% RSLogix 500 project EDINBURG_BAK719.RSS, saved by version 10.00.00.00 %
PROJECT "EDINBURG"    % processor: MicroLogix 1400 %

PROGRAM FILES
  LAD 2   12 rungs
  LAD 3   11 rungs
  LAD 4   11 rungs
  LAD 5   25 rungs
  LAD 6   8 rungs
  LAD 7   17 rungs
  LAD 8   4 rungs
  LAD 9   35 rungs
  LAD 10   2 rungs
  LAD 11   49 rungs
  LAD 12   13 rungs
  LAD 13   23 rungs

DATA FILES
  O0 OUTPUT  9 elements
  I1 INPUT  11 elements
  S2 STATUS  66 elements
  B3 BINARY  7 elements
  T4 TIMER  38 elements
  C5 COUNTER  1 elements
  R6 CONTROL  1 elements
  N7 INTEGER  40 elements
  F8 FLOAT  30 elements
  L9   1 elements
  L10   2 elements

LADDER 2
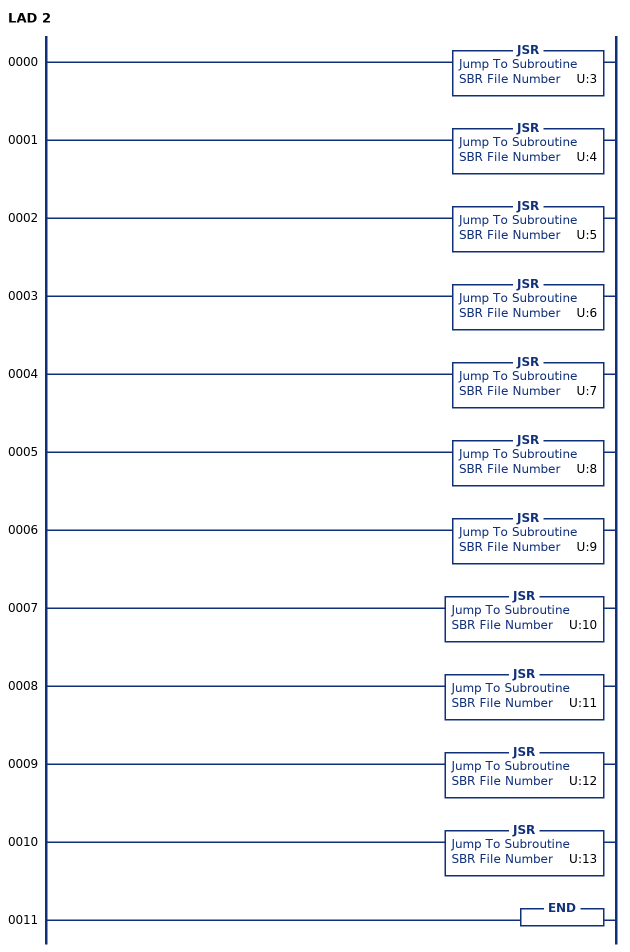
% Rung: 0 %
SOR JSR U:3 EOR
% Rung: 1 %
SOR JSR U:4 EOR
% Rung: 2 %
SOR JSR U:5 EOR
% Rung: 3 %
SOR JSR U:6 EOR
% Rung: 4 %
SOR JSR U:7 EOR
% Rung: 5 %
SOR JSR U:8 EOR
% Rung: 6 %
SOR JSR U:9 EOR
% Rung: 7 %
SOR JSR U:10 EOR
% Rung: 8 %
SOR JSR U:11 EOR
% Rung: 9 %
SOR JSR U:12 EOR
% Rung: 10 %
SOR JSR U:13 EOR
% Rung: 11 %
SOR END EOR

LADDER 3
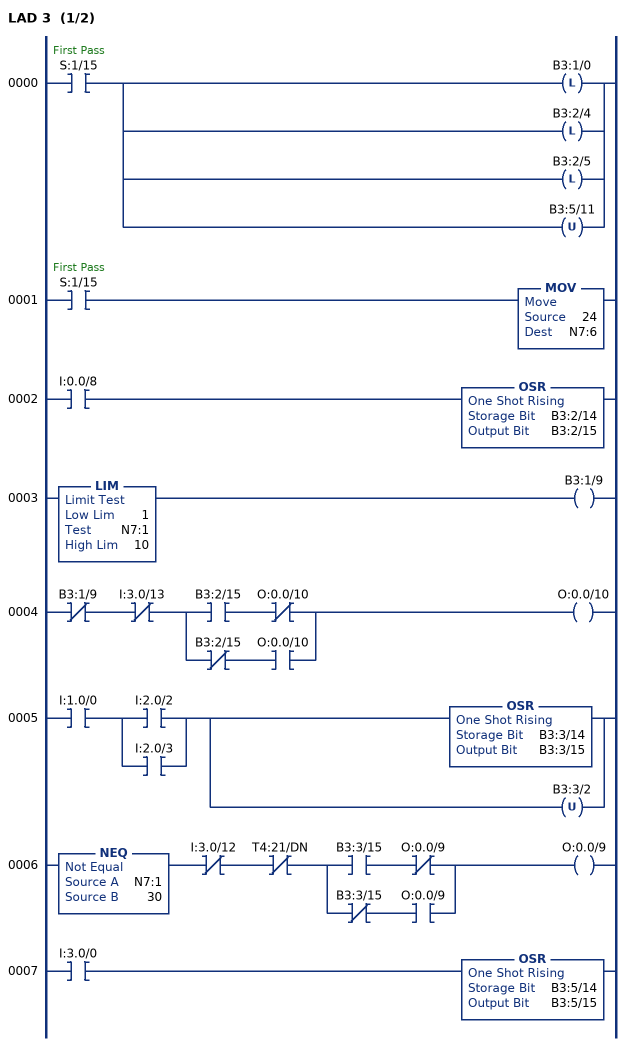
% Rung: 0 %
SOR XIC S:1/15 BST OTL B3:1/0 NXB BST OTL B3:2/4 NXB BST OTL B3:2/5 NXB OTU B3:5/11 BND BND BND EOR
%   S:1/15  "First Pass" %
% Rung: 1 %
SOR XIC S:1/15 MOV 24 N7:6 EOR
%   S:1/15  "First Pass" %
% Rung: 2 %
SOR XIC I:0.0/8 OSR B3:2/14 B3:2/15 EOR
% Rung: 3 %
SOR LIM 1 N7:1 10 OTE B3:1/9 EOR
% Rung: 4 %
SOR XIO B3:1/9 XIO I:3.0/13 BST XIC B3:2/15 XIO O:0.0/10 NXB XIO B3:2/15 XIC O:0.0/10 BND OTE O:0.0/10 EOR
% Rung: 5 %
SOR XIC I:1.0/0 BST XIC I:2.0/2 NXB XIC I:2.0/3 BND BST OSR B3:3/14 B3:3/15 NXB OTU B3:3/2 BND EOR
% Rung: 6 %
SOR NEQ N7:1 30 XIO I:3.0/12 XIO T4:21/DN BST XIC B3:3/15 XIO O:0.0/9 NXB XIO B3:3/15 XIC O:0.0/9 BND OTE O:0.0/9 EOR
% Rung: 7 %
SOR XIC I:3.0/0 OSR B3:5/14 B3:5/15 EOR

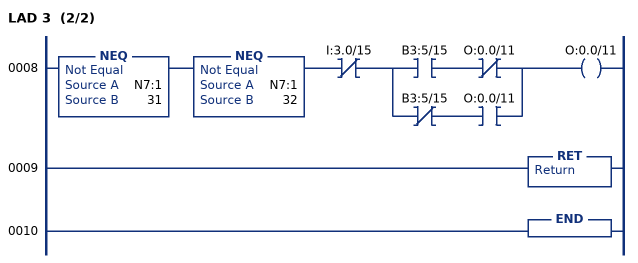
% Rung: 8 %
SOR NEQ N7:1 31 NEQ N7:1 32 XIO I:3.0/15 BST XIC B3:5/15 XIO O:0.0/11 NXB XIO B3:5/15 XIC O:0.0/11 BND OTE O:0.0/11 EOR
% Rung: 9 %
SOR RET EOR
% Rung: 10 %
SOR END EOR

LADDER 4
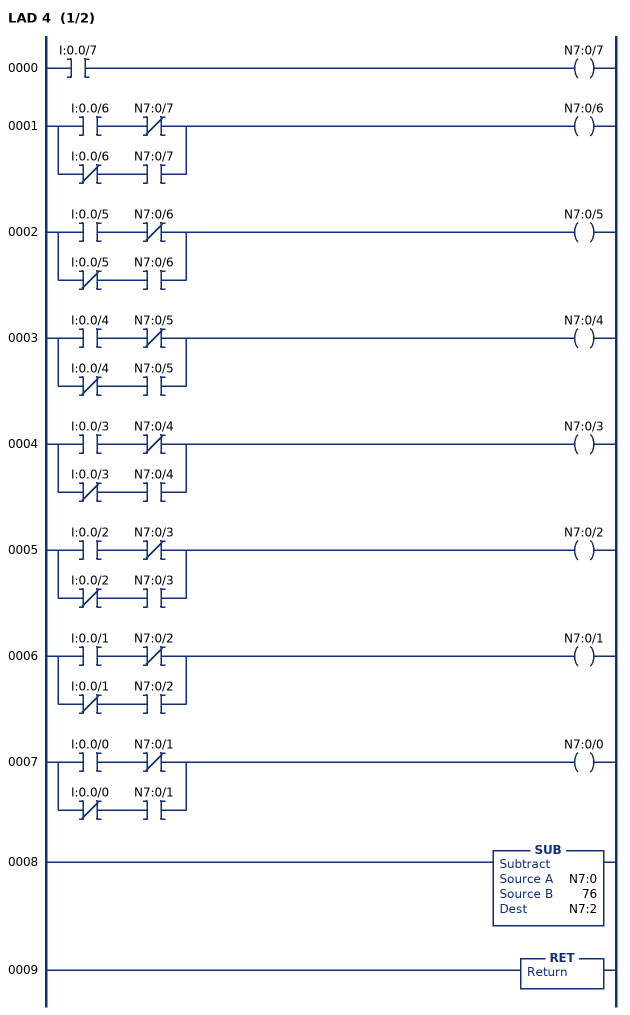
% Rung: 0 %
SOR XIC I:0.0/7 OTE N7:0/7 EOR
% Rung: 1 %
SOR BST XIC I:0.0/6 XIO N7:0/7 NXB XIO I:0.0/6 XIC N7:0/7 BND OTE N7:0/6 EOR
% Rung: 2 %
SOR BST XIC I:0.0/5 XIO N7:0/6 NXB XIO I:0.0/5 XIC N7:0/6 BND OTE N7:0/5 EOR
% Rung: 3 %
SOR BST XIC I:0.0/4 XIO N7:0/5 NXB XIO I:0.0/4 XIC N7:0/5 BND OTE N7:0/4 EOR
% Rung: 4 %
SOR BST XIC I:0.0/3 XIO N7:0/4 NXB XIO I:0.0/3 XIC N7:0/4 BND OTE N7:0/3 EOR
% Rung: 5 %
SOR BST XIC I:0.0/2 XIO N7:0/3 NXB XIO I:0.0/2 XIC N7:0/3 BND OTE N7:0/2 EOR
% Rung: 6 %
SOR BST XIC I:0.0/1 XIO N7:0/2 NXB XIO I:0.0/1 XIC N7:0/2 BND OTE N7:0/1 EOR
% Rung: 7 %
SOR BST XIC I:0.0/0 XIO N7:0/1 NXB XIO I:0.0/0 XIC N7:0/1 BND OTE N7:0/0 EOR
% Rung: 8 %
SOR SUB N7:0 76 N7:2 EOR
% Rung: 9 %
SOR RET EOR

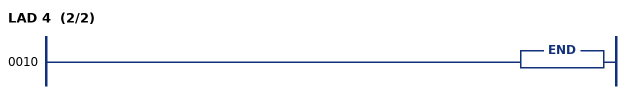
% Rung: 10 %
SOR END EOR

LADDER 5
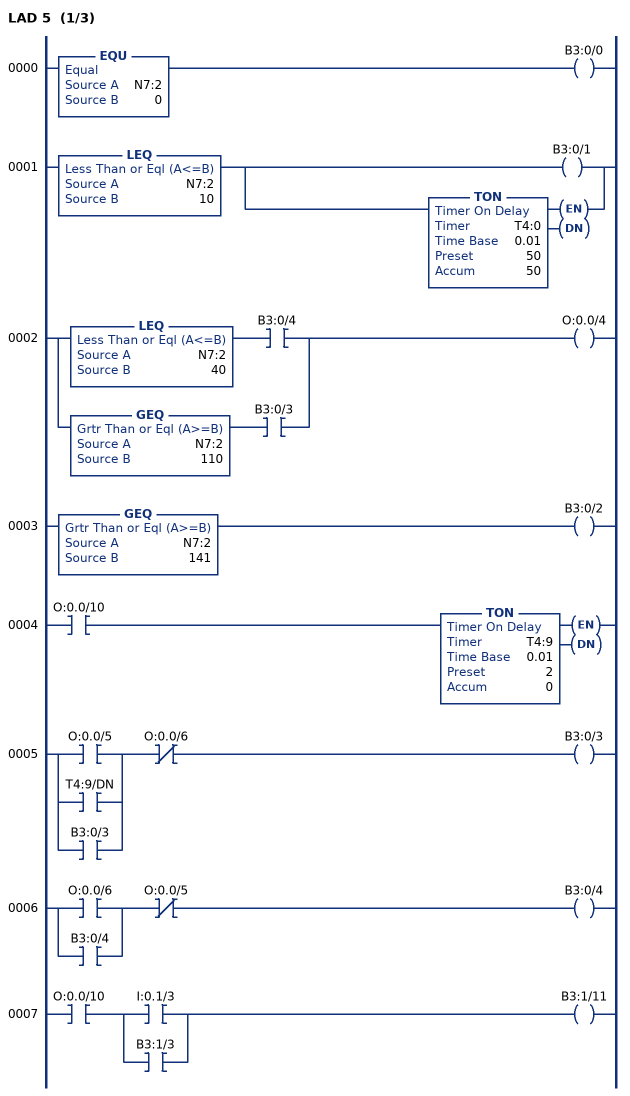
% Rung: 0 %
SOR EQU N7:2 0 OTE B3:0/0 EOR
% Rung: 1 %
SOR LEQ N7:2 10 BST OTE B3:0/1 NXB TON T4:0 0.01 50 50 BND EOR
% Rung: 2 %
SOR BST LEQ N7:2 40 XIC B3:0/4 NXB GEQ N7:2 110 XIC B3:0/3 BND OTE O:0.0/4 EOR
% Rung: 3 %
SOR GEQ N7:2 141 OTE B3:0/2 EOR
% Rung: 4 %
SOR XIC O:0.0/10 TON T4:9 0.01 2 0 EOR
% Rung: 5 %
SOR BST XIC O:0.0/5 NXB XIC T4:9/DN NXB XIC B3:0/3 BND XIO O:0.0/6 OTE B3:0/3 EOR
% Rung: 6 %
SOR BST XIC O:0.0/6 NXB XIC B3:0/4 BND XIO O:0.0/5 OTE B3:0/4 EOR
% Rung: 7 %
SOR XIC O:0.0/10 BST XIC I:0.1/3 NXB XIC B3:1/3 BND OTE B3:1/11 EOR

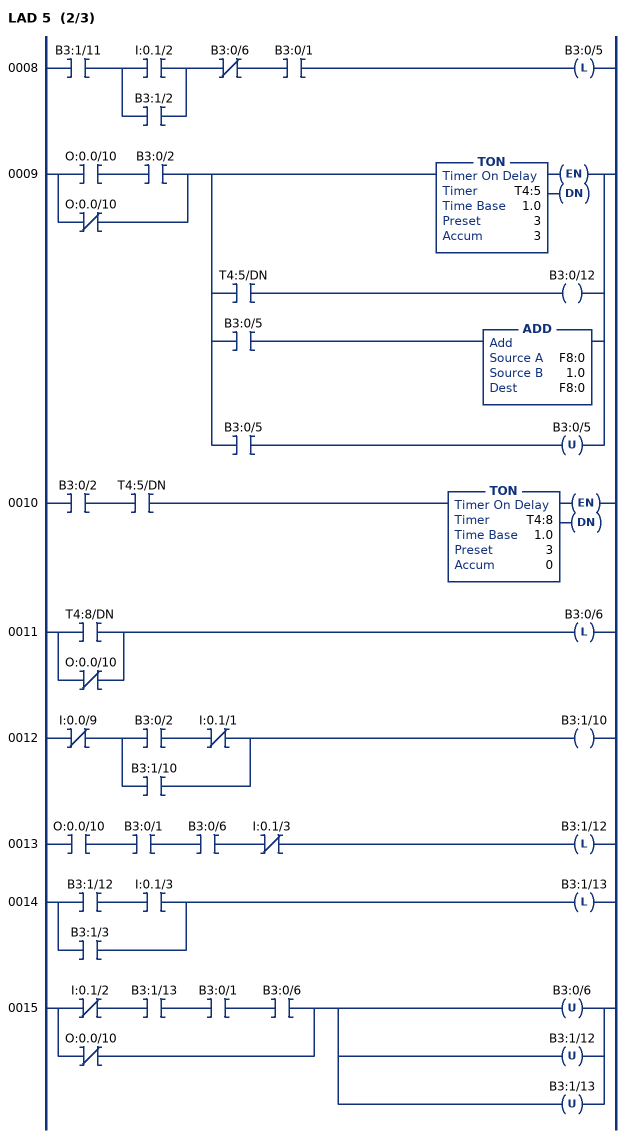
% Rung: 8 %
SOR XIC B3:1/11 BST XIC I:0.1/2 NXB XIC B3:1/2 BND XIO B3:0/6 XIC B3:0/1 OTL B3:0/5 EOR
% Rung: 9 %
SOR BST XIC O:0.0/10 XIC B3:0/2 NXB XIO O:0.0/10 BND BST TON T4:5 1.0 3 3 NXB XIC T4:5/DN OTE B3:0/12 NXB BST XIC B3:0/5 ADD F8:0 1.0 F8:0 NXB XIC B3:0/5 OTU B3:0/5 BND BND EOR
% Rung: 10 %
SOR XIC B3:0/2 XIC T4:5/DN TON T4:8 1.0 3 0 EOR
% Rung: 11 %
SOR BST XIC T4:8/DN NXB XIO O:0.0/10 BND OTL B3:0/6 EOR
% Rung: 12 %
SOR XIO I:0.0/9 BST XIC B3:0/2 XIO I:0.1/1 NXB XIC B3:1/10 BND OTE B3:1/10 EOR
% Rung: 13 %
SOR XIC O:0.0/10 XIC B3:0/1 XIC B3:0/6 XIO I:0.1/3 OTL B3:1/12 EOR
% Rung: 14 %
SOR BST XIC B3:1/12 XIC I:0.1/3 NXB XIC B3:1/3 BND OTL B3:1/13 EOR
% Rung: 15 %
SOR BST XIO I:0.1/2 XIC B3:1/13 XIC B3:0/1 XIC B3:0/6 NXB XIO O:0.0/10 BND BST OTU B3:0/6 NXB BST OTU B3:1/12 NXB OTU B3:1/13 BND BND EOR

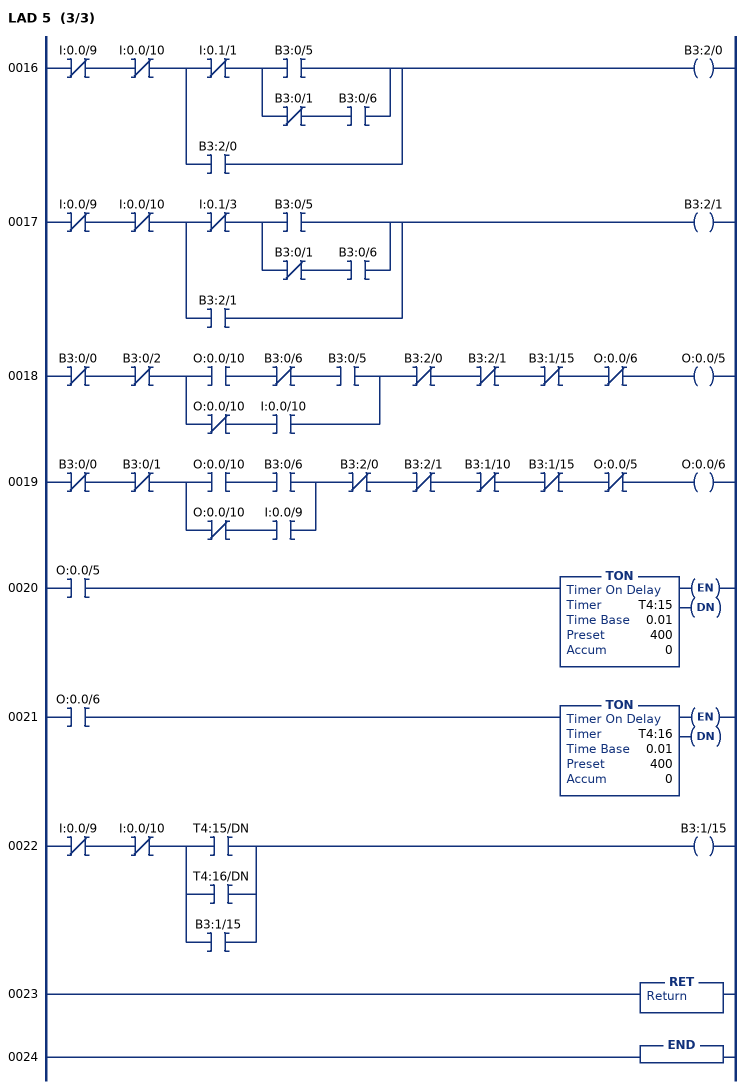
% Rung: 16 %
SOR XIO I:0.0/9 XIO I:0.0/10 BST XIO I:0.1/1 BST XIC B3:0/5 NXB XIO B3:0/1 XIC B3:0/6 BND NXB XIC B3:2/0 BND OTE B3:2/0 EOR
% Rung: 17 %
SOR XIO I:0.0/9 XIO I:0.0/10 BST XIO I:0.1/3 BST XIC B3:0/5 NXB XIO B3:0/1 XIC B3:0/6 BND NXB XIC B3:2/1 BND OTE B3:2/1 EOR
% Rung: 18 %
SOR XIO B3:0/0 XIO B3:0/2 BST XIC O:0.0/10 XIO B3:0/6 XIC B3:0/5 NXB XIO O:0.0/10 XIC I:0.0/10 BND XIO B3:2/0 XIO B3:2/1 XIO B3:1/15 XIO O:0.0/6 OTE O:0.0/5 EOR
% Rung: 19 %
SOR XIO B3:0/0 XIO B3:0/1 BST XIC O:0.0/10 XIC B3:0/6 NXB XIO O:0.0/10 XIC I:0.0/9 BND XIO B3:2/0 XIO B3:2/1 XIO B3:1/10 XIO B3:1/15 XIO O:0.0/5 OTE O:0.0/6 EOR
% Rung: 20 %
SOR XIC O:0.0/5 TON T4:15 0.01 400 0 EOR
% Rung: 21 %
SOR XIC O:0.0/6 TON T4:16 0.01 400 0 EOR
% Rung: 22 %
SOR XIO I:0.0/9 XIO I:0.0/10 BST BST XIC T4:15/DN NXB XIC T4:16/DN BND NXB XIC B3:1/15 BND OTE B3:1/15 EOR
% Rung: 23 %
SOR RET EOR
% Rung: 24 %
SOR END EOR

LADDER 6
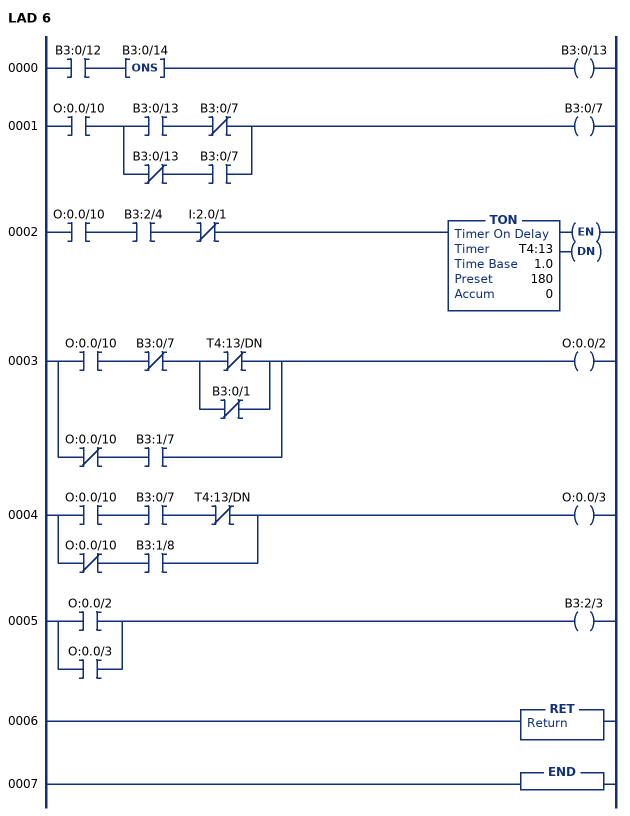
% Rung: 0 %
SOR XIC B3:0/12 ONS B3:0/14 OTE B3:0/13 EOR
% Rung: 1 %
SOR XIC O:0.0/10 BST XIC B3:0/13 XIO B3:0/7 NXB XIO B3:0/13 XIC B3:0/7 BND OTE B3:0/7 EOR
% Rung: 2 %
SOR XIC O:0.0/10 XIC B3:2/4 XIO I:2.0/1 TON T4:13 1.0 180 0 EOR
% Rung: 3 %
SOR BST XIC O:0.0/10 XIO B3:0/7 BST XIO T4:13/DN NXB XIO B3:0/1 BND NXB XIO O:0.0/10 XIC B3:1/7 BND OTE O:0.0/2 EOR
% Rung: 4 %
SOR BST XIC O:0.0/10 XIC B3:0/7 XIO T4:13/DN NXB XIO O:0.0/10 XIC B3:1/8 BND OTE O:0.0/3 EOR
% Rung: 5 %
SOR BST XIC O:0.0/2 NXB XIC O:0.0/3 BND OTE B3:2/3 EOR
% Rung: 6 %
SOR RET EOR
% Rung: 7 %
SOR END EOR

LADDER 7
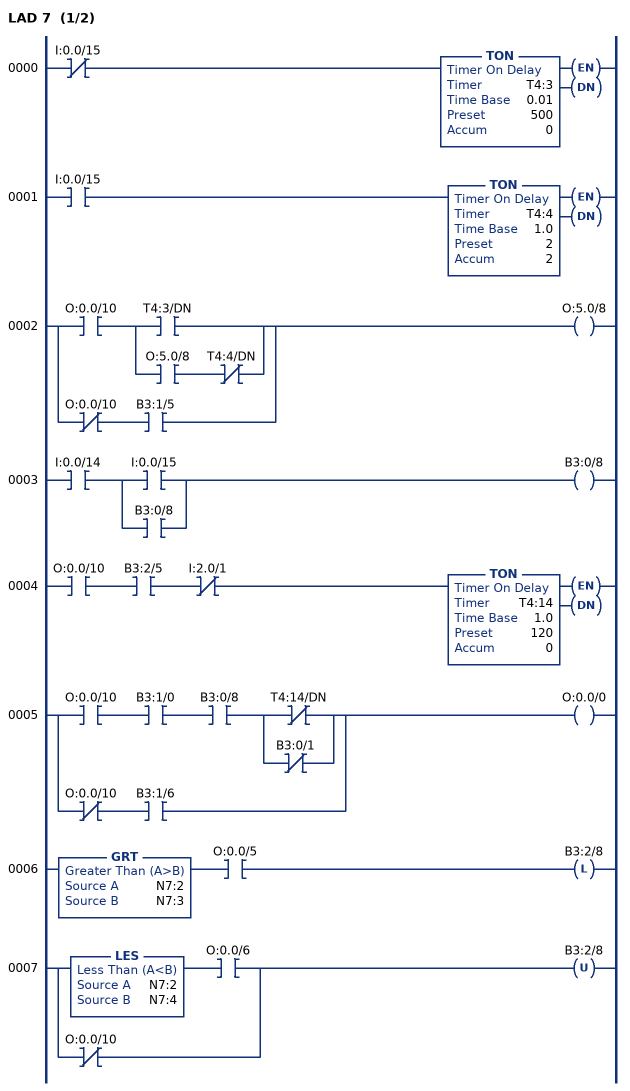
% Rung: 0 %
SOR XIO I:0.0/15 TON T4:3 0.01 500 0 EOR
% Rung: 1 %
SOR XIC I:0.0/15 TON T4:4 1.0 2 2 EOR
% Rung: 2 %
SOR BST XIC O:0.0/10 BST XIC T4:3/DN NXB XIC O:5.0/8 XIO T4:4/DN BND NXB XIO O:0.0/10 XIC B3:1/5 BND OTE O:5.0/8 EOR
% Rung: 3 %
SOR XIC I:0.0/14 BST XIC I:0.0/15 NXB XIC B3:0/8 BND OTE B3:0/8 EOR
% Rung: 4 %
SOR XIC O:0.0/10 XIC B3:2/5 XIO I:2.0/1 TON T4:14 1.0 120 0 EOR
% Rung: 5 %
SOR BST XIC O:0.0/10 XIC B3:1/0 XIC B3:0/8 BST XIO T4:14/DN NXB XIO B3:0/1 BND NXB XIO O:0.0/10 XIC B3:1/6 BND OTE O:0.0/0 EOR
% Rung: 6 %
SOR GRT N7:2 N7:3 XIC O:0.0/5 OTL B3:2/8 EOR
% Rung: 7 %
SOR BST LES N7:2 N7:4 XIC O:0.0/6 NXB XIO O:0.0/10 BND OTU B3:2/8 EOR

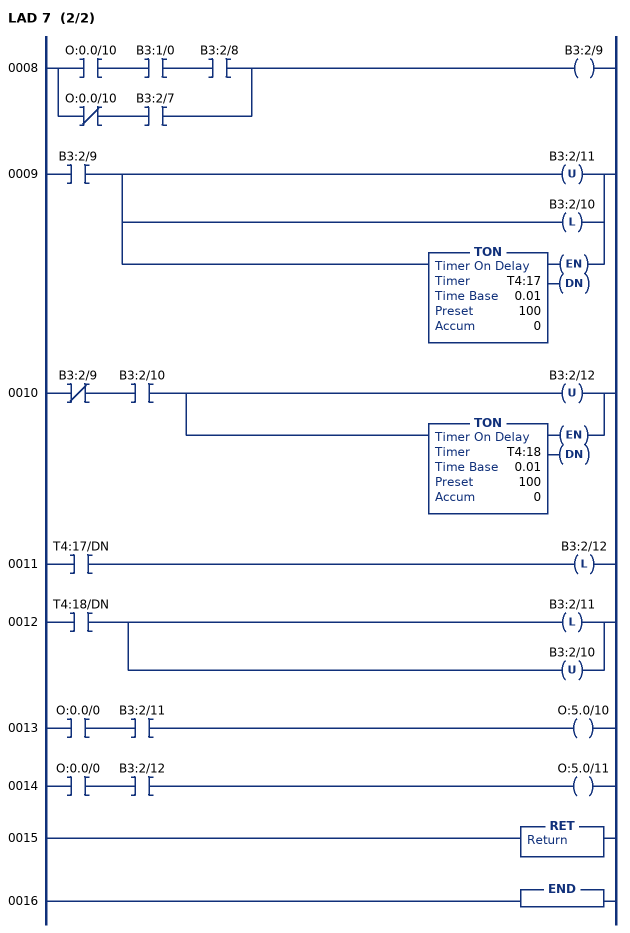
% Rung: 8 %
SOR BST XIC O:0.0/10 XIC B3:1/0 XIC B3:2/8 NXB XIO O:0.0/10 XIC B3:2/7 BND OTE B3:2/9 EOR
% Rung: 9 %
SOR XIC B3:2/9 BST OTU B3:2/11 NXB BST OTL B3:2/10 NXB TON T4:17 0.01 100 0 BND BND EOR
% Rung: 10 %
SOR XIO B3:2/9 XIC B3:2/10 BST OTU B3:2/12 NXB TON T4:18 0.01 100 0 BND EOR
% Rung: 11 %
SOR XIC T4:17/DN OTL B3:2/12 EOR
% Rung: 12 %
SOR XIC T4:18/DN BST OTL B3:2/11 NXB OTU B3:2/10 BND EOR
% Rung: 13 %
SOR XIC O:0.0/0 XIC B3:2/11 OTE O:5.0/10 EOR
% Rung: 14 %
SOR XIC O:0.0/0 XIC B3:2/12 OTE O:5.0/11 EOR
% Rung: 15 %
SOR RET EOR
% Rung: 16 %
SOR END EOR

LADDER 8
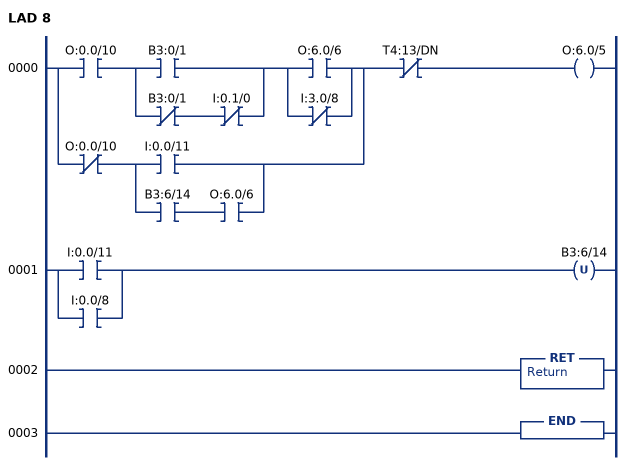
% Rung: 0 %
SOR BST XIC O:0.0/10 BST XIC B3:0/1 NXB XIO B3:0/1 XIO I:0.1/0 BND BST XIC O:6.0/6 NXB XIO I:3.0/8 BND NXB XIO O:0.0/10 BST XIC I:0.0/11 NXB XIC B3:6/14 XIC O:6.0/6 BND BND XIO T4:13/DN OTE O:6.0/5 EOR
% Rung: 1 %
SOR BST XIC I:0.0/11 NXB XIC I:0.0/8 BND OTU B3:6/14 EOR
% Rung: 2 %
SOR RET EOR
% Rung: 3 %
SOR END EOR

LADDER 9
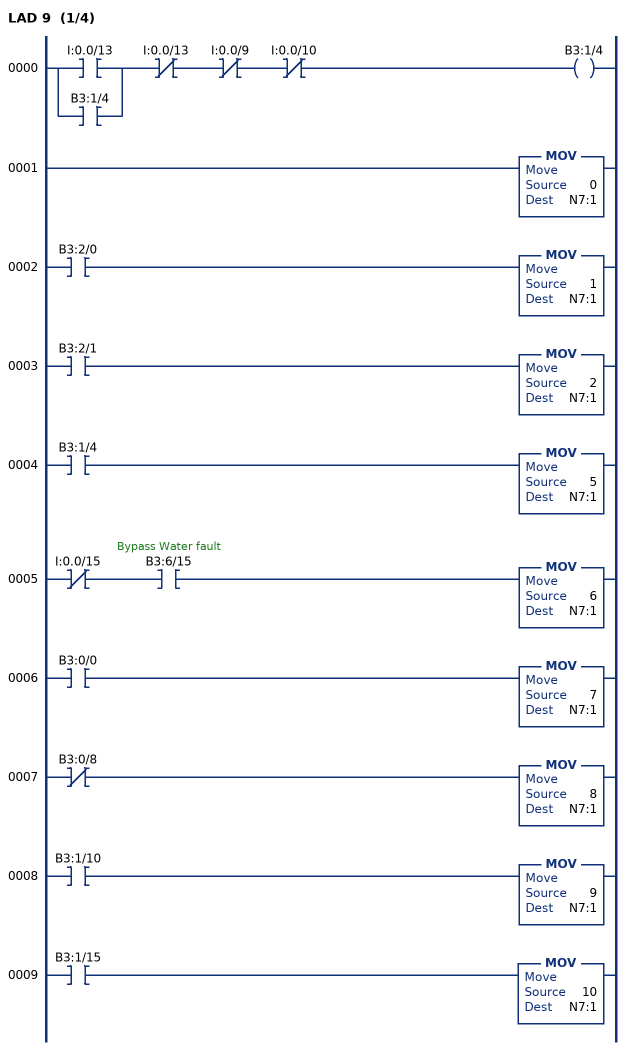
% Rung: 0 %
SOR BST XIC I:0.0/13 NXB XIC B3:1/4 BND XIO I:0.0/13 XIO I:0.0/9 XIO I:0.0/10 OTE B3:1/4 EOR
% Rung: 1 %
SOR MOV 0 N7:1 EOR
% Rung: 2 %
SOR XIC B3:2/0 MOV 1 N7:1 EOR
% Rung: 3 %
SOR XIC B3:2/1 MOV 2 N7:1 EOR
% Rung: 4 %
SOR XIC B3:1/4 MOV 5 N7:1 EOR
% Rung: 5 %
SOR XIO I:0.0/15 XIC B3:6/15 MOV 6 N7:1 EOR
%   B3:6/15  "Bypass Water fault" %
% Rung: 6 %
SOR XIC B3:0/0 MOV 7 N7:1 EOR
% Rung: 7 %
SOR XIO B3:0/8 MOV 8 N7:1 EOR
% Rung: 8 %
SOR XIC B3:1/10 MOV 9 N7:1 EOR
% Rung: 9 %
SOR XIC B3:1/15 MOV 10 N7:1 EOR

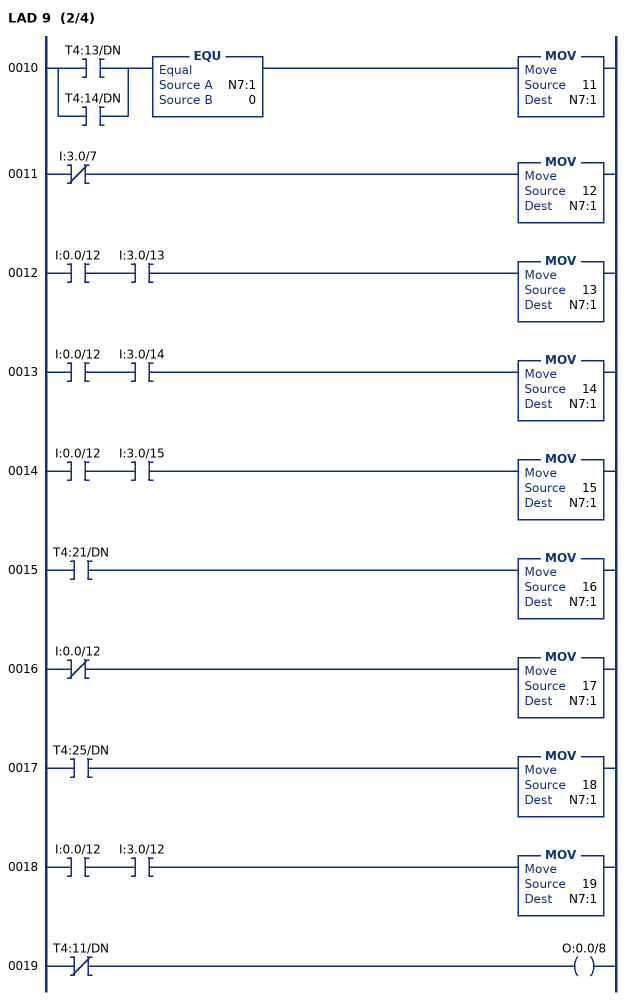
% Rung: 10 %
SOR BST XIC T4:13/DN NXB XIC T4:14/DN BND EQU N7:1 0 MOV 11 N7:1 EOR
% Rung: 11 %
SOR XIO I:3.0/7 MOV 12 N7:1 EOR
% Rung: 12 %
SOR XIC I:0.0/12 XIC I:3.0/13 MOV 13 N7:1 EOR
% Rung: 13 %
SOR XIC I:0.0/12 XIC I:3.0/14 MOV 14 N7:1 EOR
% Rung: 14 %
SOR XIC I:0.0/12 XIC I:3.0/15 MOV 15 N7:1 EOR
% Rung: 15 %
SOR XIC T4:21/DN MOV 16 N7:1 EOR
% Rung: 16 %
SOR XIO I:0.0/12 MOV 17 N7:1 EOR
% Rung: 17 %
SOR XIC T4:25/DN MOV 18 N7:1 EOR
% Rung: 18 %
SOR XIC I:0.0/12 XIC I:3.0/12 MOV 19 N7:1 EOR
% Rung: 19 %
SOR XIO T4:11/DN OTE O:0.0/8 EOR

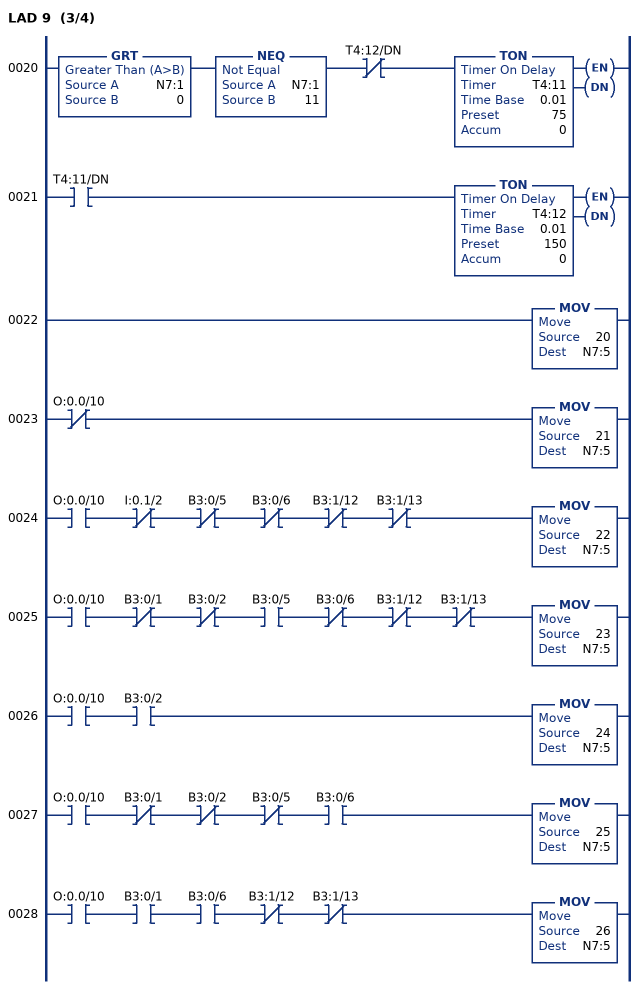
% Rung: 20 %
SOR GRT N7:1 0 NEQ N7:1 11 XIO T4:12/DN TON T4:11 0.01 75 0 EOR
% Rung: 21 %
SOR XIC T4:11/DN TON T4:12 0.01 150 0 EOR
% Rung: 22 %
SOR MOV 20 N7:5 EOR
% Rung: 23 %
SOR XIO O:0.0/10 MOV 21 N7:5 EOR
% Rung: 24 %
SOR XIC O:0.0/10 XIO I:0.1/2 XIO B3:0/5 XIO B3:0/6 XIO B3:1/12 XIO B3:1/13 MOV 22 N7:5 EOR
% Rung: 25 %
SOR XIC O:0.0/10 XIO B3:0/1 XIO B3:0/2 XIC B3:0/5 XIO B3:0/6 XIO B3:1/12 XIO B3:1/13 MOV 23 N7:5 EOR
% Rung: 26 %
SOR XIC O:0.0/10 XIC B3:0/2 MOV 24 N7:5 EOR
% Rung: 27 %
SOR XIC O:0.0/10 XIO B3:0/1 XIO B3:0/2 XIO B3:0/5 XIC B3:0/6 MOV 25 N7:5 EOR
% Rung: 28 %
SOR XIC O:0.0/10 XIC B3:0/1 XIC B3:0/6 XIO B3:1/12 XIO B3:1/13 MOV 26 N7:5 EOR

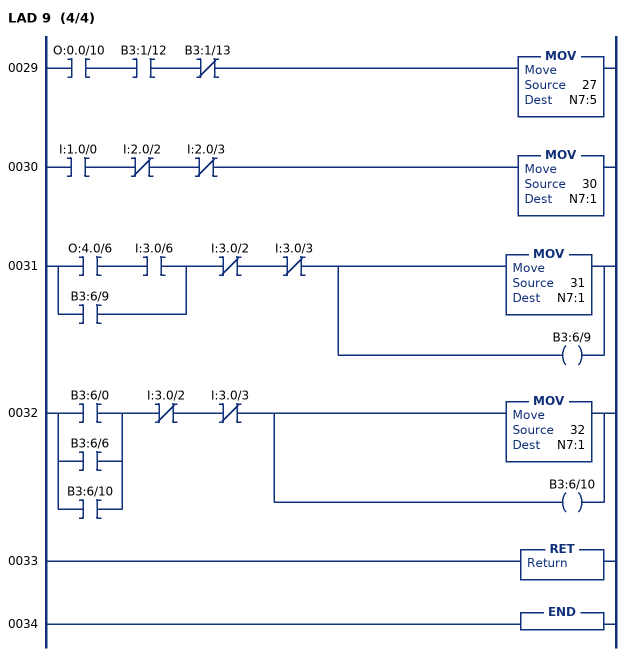
% Rung: 29 %
SOR XIC O:0.0/10 XIC B3:1/12 XIO B3:1/13 MOV 27 N7:5 EOR
% Rung: 30 %
SOR XIC I:1.0/0 XIO I:2.0/2 XIO I:2.0/3 MOV 30 N7:1 EOR
% Rung: 31 %
SOR BST XIC O:4.0/6 XIC I:3.0/6 NXB XIC B3:6/9 BND XIO I:3.0/2 XIO I:3.0/3 BST MOV 31 N7:1 NXB OTE B3:6/9 BND EOR
% Rung: 32 %
SOR BST BST XIC B3:6/0 NXB XIC B3:6/6 BND NXB XIC B3:6/10 BND XIO I:3.0/2 XIO I:3.0/3 BST MOV 32 N7:1 NXB OTE B3:6/10 BND EOR
% Rung: 33 %
SOR RET EOR
% Rung: 34 %
SOR END EOR

LADDER 10
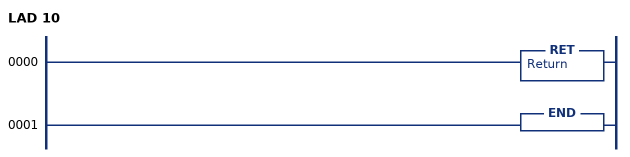
% Rung: 0 %
SOR RET EOR
% Rung: 1 %
SOR END EOR

LADDER 11
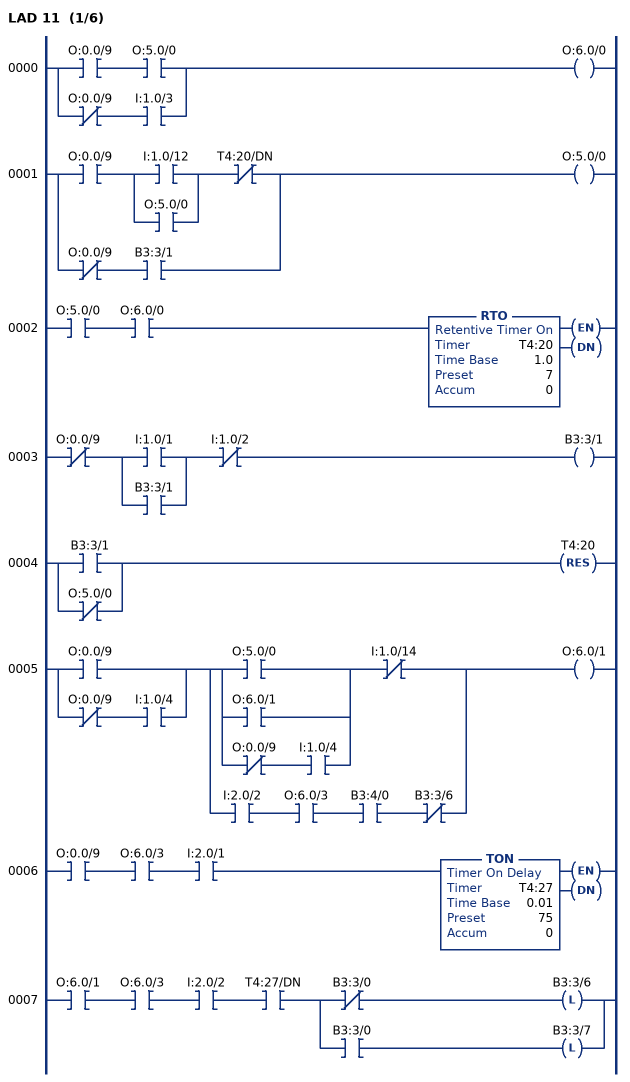
% Rung: 0 %
SOR BST XIC O:0.0/9 XIC O:5.0/0 NXB XIO O:0.0/9 XIC I:1.0/3 BND OTE O:6.0/0 EOR
% Rung: 1 %
SOR BST XIC O:0.0/9 BST XIC I:1.0/12 NXB XIC O:5.0/0 BND XIO T4:20/DN NXB XIO O:0.0/9 XIC B3:3/1 BND OTE O:5.0/0 EOR
% Rung: 2 %
SOR XIC O:5.0/0 XIC O:6.0/0 RTO T4:20 1.0 7 0 EOR
% Rung: 3 %
SOR XIO O:0.0/9 BST XIC I:1.0/1 NXB XIC B3:3/1 BND XIO I:1.0/2 OTE B3:3/1 EOR
% Rung: 4 %
SOR BST XIC B3:3/1 NXB XIO O:5.0/0 BND RES T4:20 EOR
% Rung: 5 %
SOR BST XIC O:0.0/9 NXB XIO O:0.0/9 XIC I:1.0/4 BND BST BST XIC O:5.0/0 NXB BST XIC O:6.0/1 NXB XIO O:0.0/9 XIC I:1.0/4 BND BND XIO I:1.0/14 NXB XIC I:2.0/2 XIC O:6.0/3 XIC B3:4/0 XIO B3:3/6 BND OTE O:6.0/1 EOR
% Rung: 6 %
SOR XIC O:0.0/9 XIC O:6.0/3 XIC I:2.0/1 TON T4:27 0.01 75 0 EOR
% Rung: 7 %
SOR XIC O:6.0/1 XIC O:6.0/3 XIC I:2.0/2 XIC T4:27/DN BST XIO B3:3/0 OTL B3:3/6 NXB XIC B3:3/0 OTL B3:3/7 BND EOR

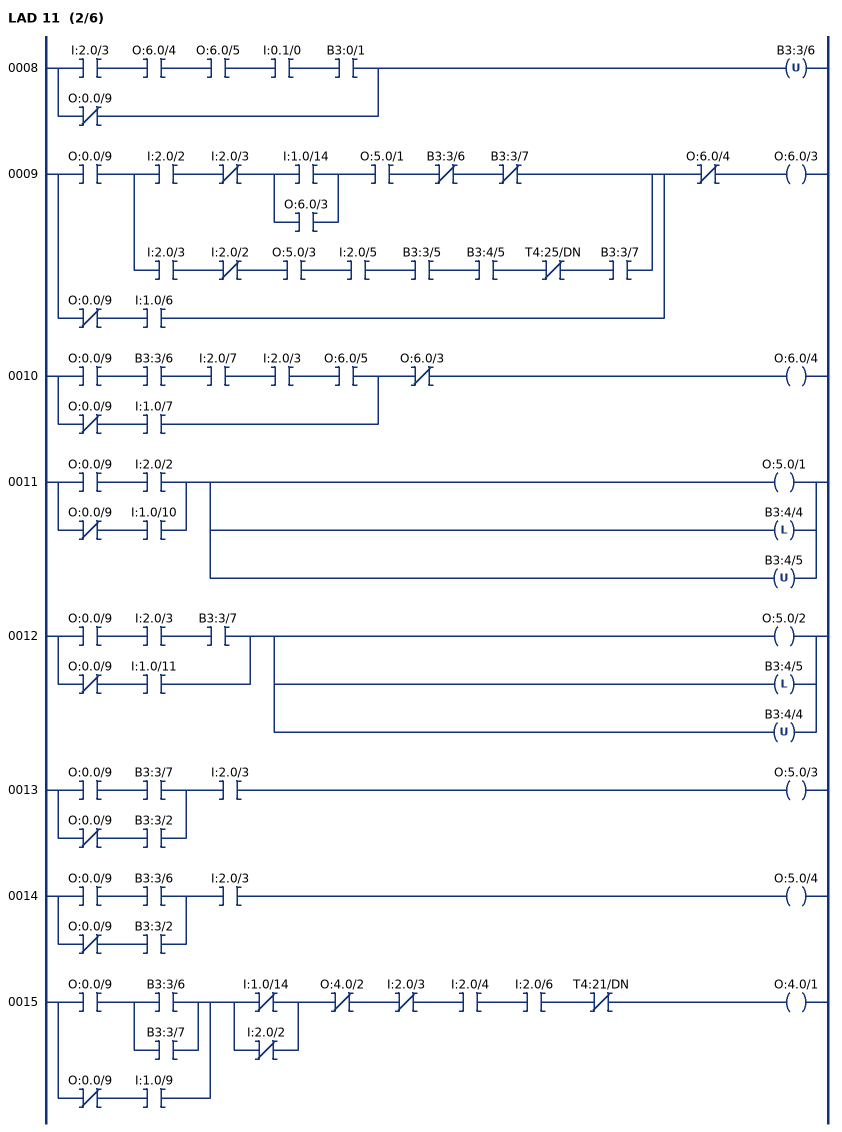
% Rung: 8 %
SOR BST XIC I:2.0/3 XIC O:6.0/4 XIC O:6.0/5 XIC I:0.1/0 XIC B3:0/1 NXB XIO O:0.0/9 BND OTU B3:3/6 EOR
% Rung: 9 %
SOR BST XIC O:0.0/9 BST XIC I:2.0/2 XIO I:2.0/3 BST XIC I:1.0/14 NXB XIC O:6.0/3 BND XIC O:5.0/1 XIO B3:3/6 XIO B3:3/7 NXB XIC I:2.0/3 XIO I:2.0/2 XIC O:5.0/3 XIC I:2.0/5 XIC B3:3/5 XIC B3:4/5 XIO T4:25/DN XIC B3:3/7 BND NXB XIO O:0.0/9 XIC I:1.0/6 BND XIO O:6.0/4 OTE O:6.0/3 EOR
% Rung: 10 %
SOR BST XIC O:0.0/9 XIC B3:3/6 XIC I:2.0/7 XIC I:2.0/3 XIC O:6.0/5 NXB XIO O:0.0/9 XIC I:1.0/7 BND XIO O:6.0/3 OTE O:6.0/4 EOR
% Rung: 11 %
SOR BST XIC O:0.0/9 XIC I:2.0/2 NXB XIO O:0.0/9 XIC I:1.0/10 BND BST OTE O:5.0/1 NXB BST OTL B3:4/4 NXB OTU B3:4/5 BND BND EOR
% Rung: 12 %
SOR BST XIC O:0.0/9 XIC I:2.0/3 XIC B3:3/7 NXB XIO O:0.0/9 XIC I:1.0/11 BND BST OTE O:5.0/2 NXB BST OTL B3:4/5 NXB OTU B3:4/4 BND BND EOR
% Rung: 13 %
SOR BST XIC O:0.0/9 XIC B3:3/7 NXB XIO O:0.0/9 XIC B3:3/2 BND XIC I:2.0/3 OTE O:5.0/3 EOR
% Rung: 14 %
SOR BST XIC O:0.0/9 XIC B3:3/6 NXB XIO O:0.0/9 XIC B3:3/2 BND XIC I:2.0/3 OTE O:5.0/4 EOR
% Rung: 15 %
SOR BST XIC O:0.0/9 BST XIC B3:3/6 NXB XIC B3:3/7 BND NXB XIO O:0.0/9 XIC I:1.0/9 BND BST XIO I:1.0/14 NXB XIO I:2.0/2 BND XIO O:4.0/2 XIO I:2.0/3 XIC I:2.0/4 XIC I:2.0/6 XIO T4:21/DN OTE O:4.0/1 EOR

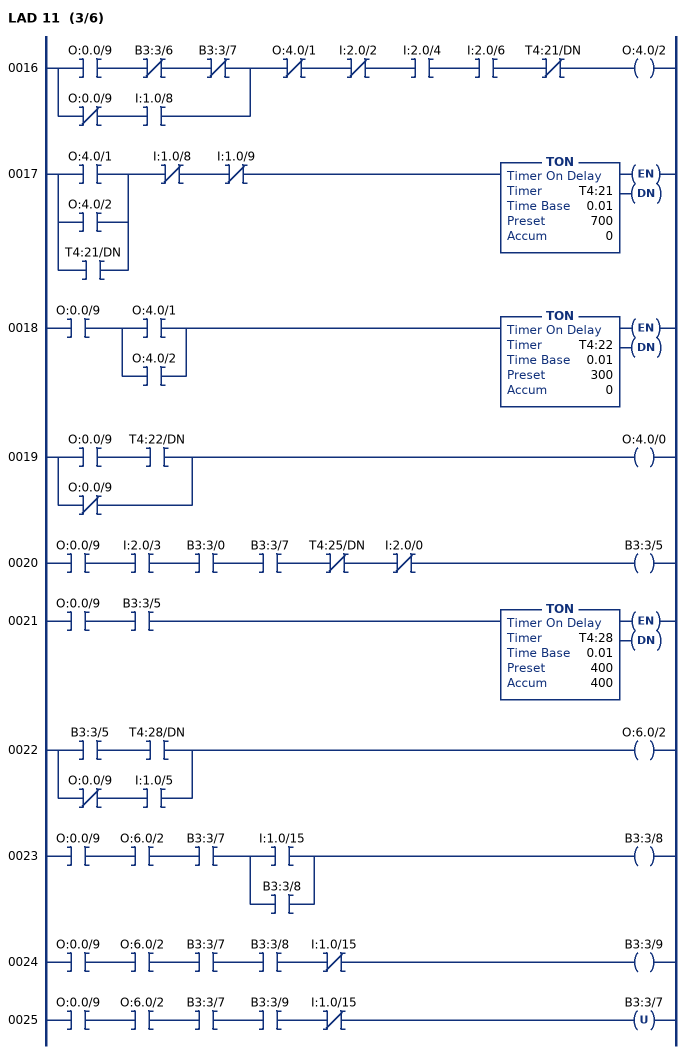
% Rung: 16 %
SOR BST XIC O:0.0/9 XIO B3:3/6 XIO B3:3/7 NXB XIO O:0.0/9 XIC I:1.0/8 BND XIO O:4.0/1 XIO I:2.0/2 XIC I:2.0/4 XIC I:2.0/6 XIO T4:21/DN OTE O:4.0/2 EOR
% Rung: 17 %
SOR BST BST XIC O:4.0/1 NXB XIC O:4.0/2 BND NXB XIC T4:21/DN BND XIO I:1.0/8 XIO I:1.0/9 TON T4:21 0.01 700 0 EOR
% Rung: 18 %
SOR XIC O:0.0/9 BST XIC O:4.0/1 NXB XIC O:4.0/2 BND TON T4:22 0.01 300 0 EOR
% Rung: 19 %
SOR BST XIC O:0.0/9 XIC T4:22/DN NXB XIO O:0.0/9 BND OTE O:4.0/0 EOR
% Rung: 20 %
SOR XIC O:0.0/9 XIC I:2.0/3 XIC B3:3/0 XIC B3:3/7 XIO T4:25/DN XIO I:2.0/0 OTE B3:3/5 EOR
% Rung: 21 %
SOR XIC O:0.0/9 XIC B3:3/5 TON T4:28 0.01 400 400 EOR
% Rung: 22 %
SOR BST XIC B3:3/5 XIC T4:28/DN NXB XIO O:0.0/9 XIC I:1.0/5 BND OTE O:6.0/2 EOR
% Rung: 23 %
SOR XIC O:0.0/9 XIC O:6.0/2 XIC B3:3/7 BST XIC I:1.0/15 NXB XIC B3:3/8 BND OTE B3:3/8 EOR
% Rung: 24 %
SOR XIC O:0.0/9 XIC O:6.0/2 XIC B3:3/7 XIC B3:3/8 XIO I:1.0/15 OTE B3:3/9 EOR
% Rung: 25 %
SOR XIC O:0.0/9 XIC O:6.0/2 XIC B3:3/7 XIC B3:3/9 XIO I:1.0/15 OTU B3:3/7 EOR

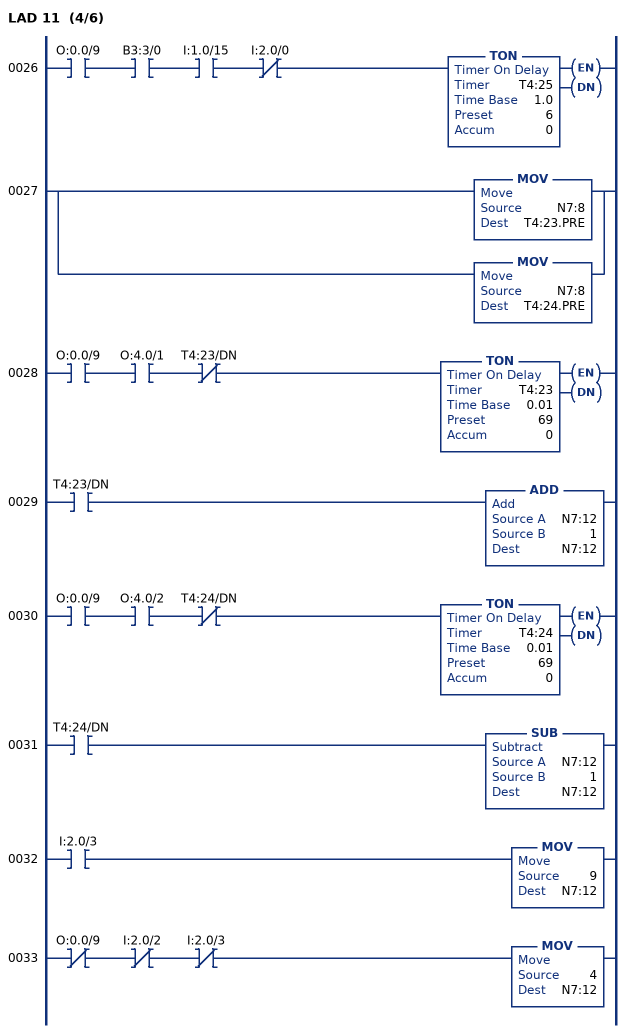
% Rung: 26 %
SOR XIC O:0.0/9 XIC B3:3/0 XIC I:1.0/15 XIO I:2.0/0 TON T4:25 1.0 6 0 EOR
% Rung: 27 %
SOR BST MOV N7:8 T4:23.PRE NXB MOV N7:8 T4:24.PRE BND EOR
% Rung: 28 %
SOR XIC O:0.0/9 XIC O:4.0/1 XIO T4:23/DN TON T4:23 0.01 69 0 EOR
% Rung: 29 %
SOR XIC T4:23/DN ADD N7:12 1 N7:12 EOR
% Rung: 30 %
SOR XIC O:0.0/9 XIC O:4.0/2 XIO T4:24/DN TON T4:24 0.01 69 0 EOR
% Rung: 31 %
SOR XIC T4:24/DN SUB N7:12 1 N7:12 EOR
% Rung: 32 %
SOR XIC I:2.0/3 MOV 9 N7:12 EOR
% Rung: 33 %
SOR XIO O:0.0/9 XIO I:2.0/2 XIO I:2.0/3 MOV 4 N7:12 EOR

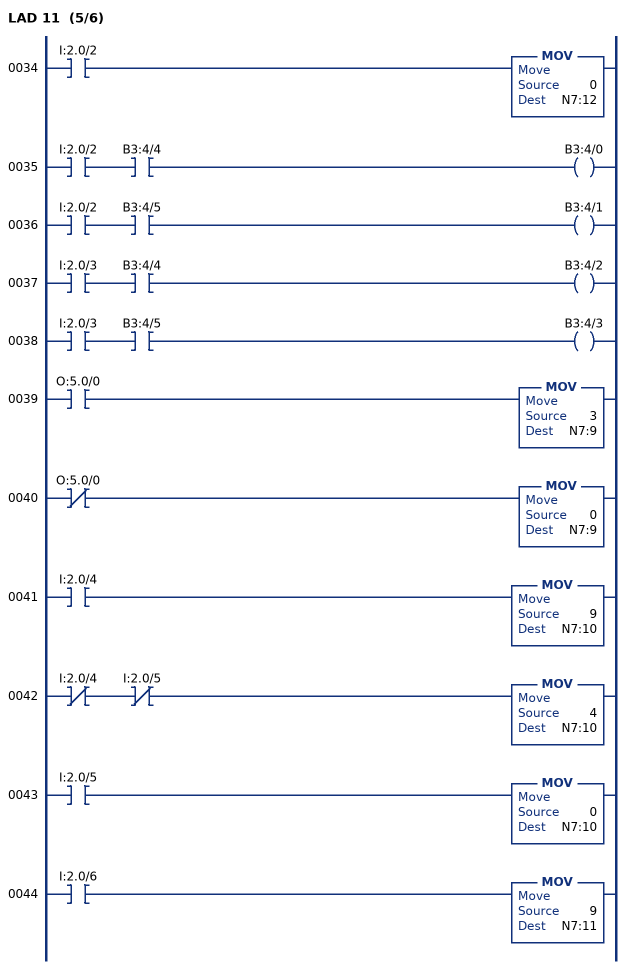
% Rung: 34 %
SOR XIC I:2.0/2 MOV 0 N7:12 EOR
% Rung: 35 %
SOR XIC I:2.0/2 XIC B3:4/4 OTE B3:4/0 EOR
% Rung: 36 %
SOR XIC I:2.0/2 XIC B3:4/5 OTE B3:4/1 EOR
% Rung: 37 %
SOR XIC I:2.0/3 XIC B3:4/4 OTE B3:4/2 EOR
% Rung: 38 %
SOR XIC I:2.0/3 XIC B3:4/5 OTE B3:4/3 EOR
% Rung: 39 %
SOR XIC O:5.0/0 MOV 3 N7:9 EOR
% Rung: 40 %
SOR XIO O:5.0/0 MOV 0 N7:9 EOR
% Rung: 41 %
SOR XIC I:2.0/4 MOV 9 N7:10 EOR
% Rung: 42 %
SOR XIO I:2.0/4 XIO I:2.0/5 MOV 4 N7:10 EOR
% Rung: 43 %
SOR XIC I:2.0/5 MOV 0 N7:10 EOR
% Rung: 44 %
SOR XIC I:2.0/6 MOV 9 N7:11 EOR

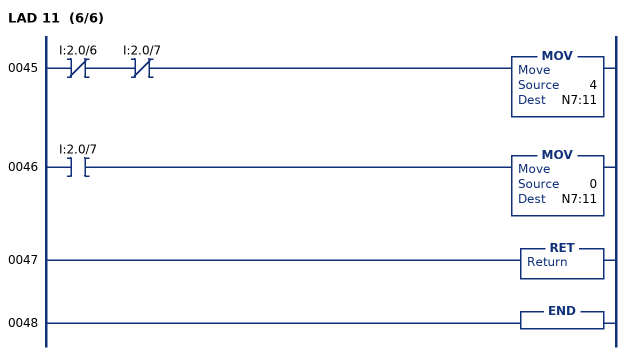
% Rung: 45 %
SOR XIO I:2.0/6 XIO I:2.0/7 MOV 4 N7:11 EOR
% Rung: 46 %
SOR XIC I:2.0/7 MOV 0 N7:11 EOR
% Rung: 47 %
SOR RET EOR
% Rung: 48 %
SOR END EOR

LADDER 12
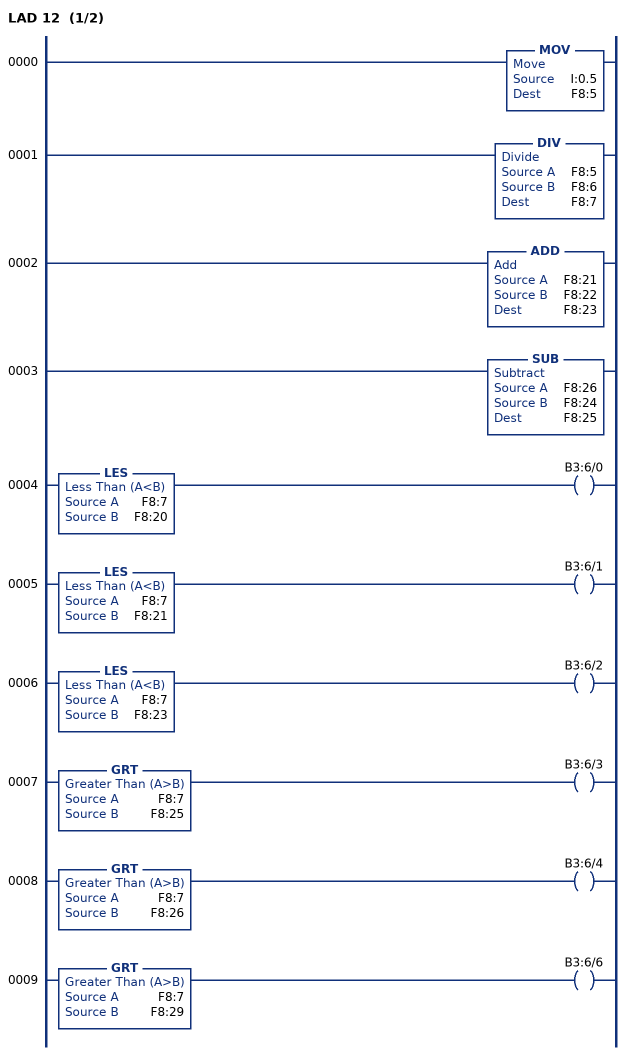
% Rung: 0 %
SOR MOV I:0.5 F8:5 EOR
% Rung: 1 %
SOR DIV F8:5 F8:6 F8:7 EOR
% Rung: 2 %
SOR ADD F8:21 F8:22 F8:23 EOR
% Rung: 3 %
SOR SUB F8:26 F8:24 F8:25 EOR
% Rung: 4 %
SOR LES F8:7 F8:20 OTE B3:6/0 EOR
% Rung: 5 %
SOR LES F8:7 F8:21 OTE B3:6/1 EOR
% Rung: 6 %
SOR LES F8:7 F8:23 OTE B3:6/2 EOR
% Rung: 7 %
SOR GRT F8:7 F8:25 OTE B3:6/3 EOR
% Rung: 8 %
SOR GRT F8:7 F8:26 OTE B3:6/4 EOR
% Rung: 9 %
SOR GRT F8:7 F8:29 OTE B3:6/6 EOR

